// Mitsubishi GX Works2 project: PLC 특수 Relay (접점)   PLC: Q03UDV

PROGRAM MAIN
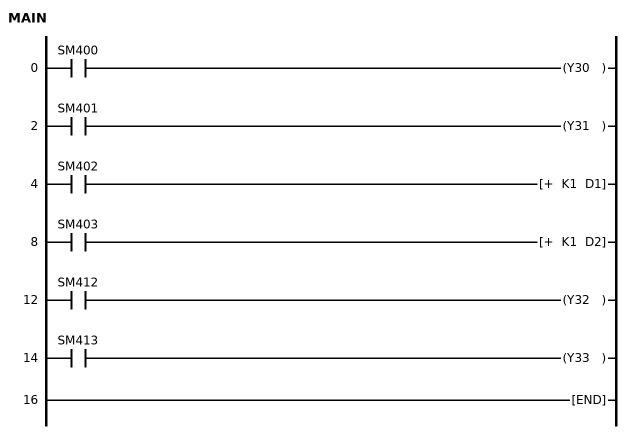
0     LD      SM400
      OUT     Y30
2     LD      SM401
      OUT     Y31
4     LD      SM402
      +       K1 D1
8     LD      SM403
      +       K1 D2
12    LD      SM412
      OUT     Y32
14    LD      SM413
      OUT     Y33
16    END
END_PROGRAM
